(* IEC 61131-3 sources: Daniele1996.github.io/AUTOMATION_AND_SOFTWARE_DESIGN_PATTERN/AUTOMATION_STUDIO/Task1/Logical/Libraries/filter_lib, 5 files *)

(* ---- Types.typ ---- *)
TYPE

END_TYPE

(* ---- BlinkFB.st ---- *)
(* TODO: Add your comment here *)
FUNCTION_BLOCK BlinkFB
	IF Clock = 0 THEN
		LED := NOT LED;
		Clock := Delay;

	ELSE
		Clock := Clock -1;
	END_IF
END_FUNCTION_BLOCK

(* ---- filter.st ---- *)
(* TODO: Add your comment here *)
FUNCTION_BLOCK filter

	IF Delay > 0 THEN
		Delay := Delay -1;
	END_IF;

	IF Delay = 0 THEN
	  DelayedSignal := Signal;
	END_IF;

	IF Signal = DelayedSignal THEN

		IF Signal THEN
			Delay := DeactivationDelay;
		ELSE
			Delay := ActivationDelay;
		END_IF;

	END_IF;
END_FUNCTION_BLOCK

(* ---- Constants.var ---- *)
VAR CONSTANT

END_VAR

(* ---- filter_lib.fun ---- *)
{REDUND_ERROR} {REDUND_UNREPLICABLE} FUNCTION_BLOCK filter (*TODO: Add your comment here*) (*$GROUP=User,$CAT=User,$GROUPICON=User.png,$CATICON=User.png*)
	VAR_INPUT
		Signal : {REDUND_UNREPLICABLE} BOOL;
		ActivationDelay : {REDUND_UNREPLICABLE} UDINT;
		DeactivationDelay : {REDUND_UNREPLICABLE} UDINT;
	END_VAR
	VAR_OUTPUT
		DelayedSignal : {REDUND_UNREPLICABLE} BOOL;
	END_VAR
	VAR
		Delay : {REDUND_UNREPLICABLE} UDINT;
	END_VAR
END_FUNCTION_BLOCK

{REDUND_ERROR} {REDUND_UNREPLICABLE} FUNCTION_BLOCK BlinkFB (*TODO: Add your comment here*) (*$GROUP=User,$CAT=User,$GROUPICON=User.png,$CATICON=User.png*)
	VAR_INPUT RETAIN
		Delay : {REDUND_UNREPLICABLE} INT := 5;
	END_VAR
	VAR_IN_OUT
		LED : BOOL;
	END_VAR
	VAR
		Clock : {REDUND_UNREPLICABLE} INT;
	END_VAR
END_FUNCTION_BLOCK
